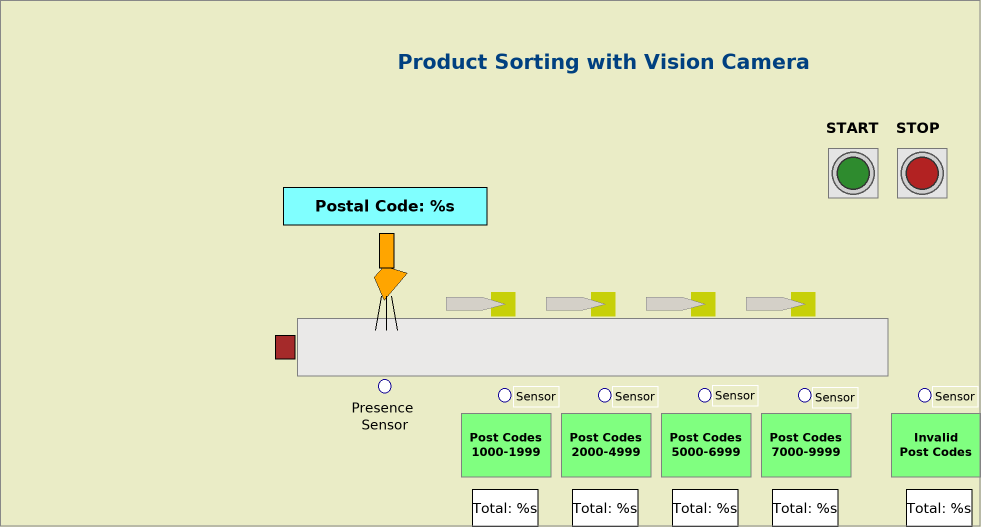
VISUALIZATION Visualization  // 981x527
    Polygon (374,277) (384,266) (407,273) (384,300), colour toggle: MAIN.Control.CameraDetect.Busy
    Rectangle (379,233 15x35)
    Rectangle (297,318 591x58), colour toggle: MAIN.Control.ConveyorMotorCmd
    Rectangle (275,335 20x24)
        p3560616238: Simulation.ProductPosition.X
        p2738717112: Simulation.ProductPosition.y
    Ellipse (378,379 13x14), colour toggle: GVL.ProductPresenceSensor
    Rectangle (491,292 24x24)
    Polygon (446,297) (482,297) (505,304) (482,310) (446,310)
        p2858320360: BOOL_TO_INT(MAIN.Control.Arm01Cmd) * 90
    Rectangle (591,292 24x24)
    Rectangle (691,292 24x24)
    Rectangle (791,292 24x24)
    Line (386,296) (386,330), invisible if: NOT MAIN.Control.CameraDetect.Busy
    Line (391,296) (397,330), invisible if: NOT MAIN.Control.CameraDetect.Busy
    Line (381,296) (375,330), invisible if: NOT MAIN.Control.CameraDetect.Busy
    Rectangle (461,413 90x64), "Post Codes 1000-1999"
    Rectangle (561,413 90x64), "Post Codes 2000-4999"
    Rectangle (661,413 90x64), "Post Codes 5000-6999"
    Rectangle (761,413 90x64), "Post Codes 7000-9999"
    Ellipse (498,388 13x14), colour toggle: GVL.PostCodeSensor01
    Rectangle (891,413 90x64), "Invalid Post Codes"
    Polygon (546,297) (582,297) (605,304) (582,310) (546,310)
        p2858320360: BOOL_TO_INT(MAIN.Control.Arm02Cmd) * 90
    Polygon (646,297) (682,297) (705,304) (682,310) (646,310)
        p2858320360: BOOL_TO_INT(MAIN.Control.Arm03Cmd) * 90
    Polygon (746,297) (782,297) (805,304) (782,310) (746,310)
        p2858320360: BOOL_TO_INT(MAIN.Control.Arm04Cmd) * 90
    Ellipse (598,388 13x14), colour toggle: GVL.PostCodeSensor02
    Ellipse (698,388 13x14), colour toggle: GVL.PostCodeSensor03
    Ellipse (798,388 13x14), colour toggle: GVL.PostCodeSensor04
    Ellipse (918,388 13x14), colour toggle: GVL.InvalidPostCodesSensor
    Rectangle (349,398 72x37), "Presence Sensor"
    Rectangle (513,386 46x21), "Sensor"
    Rectangle (612,386 46x21), "Sensor"
    Rectangle (712,385 46x21), "Sensor"
    Rectangle (812,387 46x21), "Sensor"
    Rectangle (932,386 46x21), "Sensor"
    PushSwitch (828,148 50x50), variable: GVL.StartButton, behaviour: TAP, style: Switch-PushSwitch-Green
    PushSwitch (897,148 50x50), variable: GVL.StopButton, behaviour: TAP, style: Switch-PushSwitch-Red
    RoundedRectangle (472,489 66x38), "Total: %s", text variable: MAIN.Control.PostCodeProducts01Count
    RoundedRectangle (572,489 66x38), "Total: %s", text variable: MAIN.Control.PostCodeProducts02Count
    RoundedRectangle (672,489 66x38), "Total: %s", text variable: MAIN.Control.PostCodeProducts03Count
    RoundedRectangle (772,489 66x38), "Total: %s", text variable: MAIN.Control.PostCodeProducts04Count
    RoundedRectangle (906,489 66x38), "Total: %s", text variable: MAIN.Control.InvalidPostCodeCount
    RoundedRectangle (283,187 204x38), "Postal Code: %s", text variable: MAIN.Control.ProductCode
    Rectangle (810,113 85x30), "START"
    Rectangle (885,113 66x30), "STOP"
    Rectangle (394,47 420x30), "Product Sorting with Vision Camera"
END_VISUALIZATION

(* stored: Version 1.1.0.1, ProductVersion 3.1.4024.15
   Visu Visualization: Id {96a8f8c3-d5f2-4463-8caa-fe2e7d56549c} *)
